FUNCTION_BLOCK FB_KPI_OuterLevelCounter
VAR_INPUT
	bExecute					: BOOL;			(* set TRUE to add value to buffer *)
	stCTDateTime				: ST_SYSTEM_DateTime;	(* CaseTrace date/time structure *)
	sOuterStatus				: ST_OUTER_Status;	(* Outer status *)
	aRejectCountersID			: ARRAY[0..cMAX_REJECT_REASON] OF UINT;
END_VAR
VAR_IN_OUT
	aShiftRejectCounters		: ARRAY[0..cMAX_REJECT_REASON] OF ST_LOG_RejectReasons;
	aProdRejectCounters		: ARRAY[0..cMAX_REJECT_REASON] OF ST_LOG_RejectReasons;
END_VAR
VAR_OUTPUT
	bDone					: BOOL;			(* TRUE = complete *)
END_VAR
VAR
	fbExecute					: R_TRIG;
	//nMaxIndex				: UINT;

	nRejectIndex				: T_PositiveINT;

END_VAR

(* rising edge of bExecute *)
fbExecute(CLK:= bExecute);

(* search for strBarcode in queue *)
IF fbExecute.Q = TRUE THEN

	FOR nRejectIndex := 0  TO  cMAX_REJECT_REASON DO
		IF sOuterStatus.stOACData.OuterRejectID = aRejectCountersID[nRejectIndex] THEN

			aShiftRejectCounters[nRejectIndex].nRejectCounter := aShiftRejectCounters[nRejectIndex].nRejectCounter + 1;
			aShiftRejectCounters[nRejectIndex].stLastTimeStamp := stCTDateTime.sSystemTime;

			aProdRejectCounters[nRejectIndex].nRejectCounter := aProdRejectCounters[nRejectIndex].nRejectCounter + 1;
			aProdRejectCounters[nRejectIndex].stLastTimeStamp := stCTDateTime.sSystemTime;
			EXIT;
		END_IF
	END_FOR

	bDone := TRUE;

(* bExecute has been reset *)
ELSIF bExecute = FALSE THEN

	(* reset outputs *)
	bDone := FALSE;

END_IF

END_FUNCTION_BLOCK

(* stored: Version 1.1.0.1
   POU FB_KPI_OuterLevelCounter: Id {12ad3771-0f2b-46e3-8546-9a516df63292}, SpecialFunc None *)
